(* IEC 61131-3 sources: osaicnc/, 32 files *)

(* ---- F_BitPosition.st ---- *)
(*[[
    UserText1= "V15.7",
]]*)
FUNCTION F_BitPosition : INT
(*
F ***************************************************************************************
F * File name    : F_BitPosition.st                                                     *
F * Description  : Calculate the position of a single bit into the input variable, from *
F *                1 to 15, the function give zero if more then one bit is true, if the *
F *                most significative bit is true, if all the bits are false.           *
F *                Especially thinked to convert the SW31 S_1PROMOD variable in the     *
F *                SetProcessMode function block format.                                *
F ***************************************************************************************
F * Product line : OpenControl                                                          *
F * Enviroment   : PLC Application                                                      *
F * Component    :                                                                      *
F *                                                                                     *
F * ----------------------------------------------------------------------------------- *
F *                                                                                     *
F *   Author        date        comments                                                *
F *                                                                                     *
F *   Mazzocco      19-03-10    Creation F_BitPosition                                  *
F *                                                                                     *
F * ----------------------------------------------------------------------------------- *
F *                                                                                     *
F * Input        :  iiVariable          INT                                             *
F *                     Input variable with only one bit true, except the most          *
F *                     significative bit                                               *
F *                                                                                     *
F * Return       :  INT                                                                 *
F *                     Position of a single bit into the input variable, from 1 to 15, *
F *                     the function give zero if more then one bit or the most         *
F *                     significative bit is true                                       *
F *                                                                                     *
F * Global used  :      Not used                                                        *
F *                                                                                     *
F ***************************************************************************************

	Example for program use

\* F_BitPosition function calculate the position of a single bit into the input variable, from
	1 to 15, the function give zero if more then one bit is true, if the most significative bit
	is true, if all the bits are false */
liNewValue	:= F_BitPosition(iiVariable);
*)

VAR_INPUT
	iiVariable	: int;	(* Input variable with only one bit true, except the most significative bit *)
END_VAR

case iiVariable of
	1:		F_BitPosition	:= 1;
	2:		F_BitPosition	:= 2;
	4:		F_BitPosition	:= 3;
	8:		F_BitPosition	:= 4;
	16:		F_BitPosition	:= 5;
	32:		F_BitPosition	:= 6;
	64:		F_BitPosition	:= 7;
	128:	F_BitPosition	:= 8;
	256:	F_BitPosition	:= 9;
	512:	F_BitPosition	:= 10;
	1024:	F_BitPosition	:= 11;
	2048:	F_BitPosition	:= 12;
	4096:	F_BitPosition	:= 13;
	8192:	F_BitPosition	:= 14;
	16384:	F_BitPosition	:= 15;
	-32768:	F_BitPosition	:= 16;
else
    F_BitPosition	:= 0;
end_case;

END_FUNCTION

(* ---- F_CompareArray.st ---- *)
(*[[
    UserText1= "V15.7",
]]*)
FUNCTION F_CompareArray : BOOL
(*
F ***************************************************************************************
F * File name    : F_CompareArray.st                                                    *
F * Description  : Compare two array with NUM_OF_AX fields, to check if they countain   *
F *                the same value, in the same or in different order.                   *
F ***************************************************************************************
F * Product line : OpenControl                                                          *
F * Enviroment   : PLC Application                                                      *
F * Component    :                                                                      *
F *                                                                                     *
F * ----------------------------------------------------------------------------------- *
F *                                                                                     *
F *   Author        date        comments                                                *
F *                                                                                     *
F *   Mazzocco      18-05-10    Function creation                                       *
F *                                                                                     *
F * ----------------------------------------------------------------------------------- *
F *                                                                                     *
F * Input        :  iiArray1            Array [0..NUM_OF_AX-1] of INT                   *
F *                     First array                                                     *
F *                                                                                     *
F *                 iiArray2            Array [0..NUM_OF_AX-1] of INT                   *
F *                     Second array                                                    *
F *                                                                                     *
F * Return       :  BOOL                                                                *
F *                     True value if both arrays countain the same value in any order  *
F *                                                                                     *
F * Global used  :      Not used                                                        *
F *                                                                                     *
F ***************************************************************************************

	Example for program use

\* Compare two array with NUM_OF_AX fields, to check if they countain the same value, in the
	same or in different order */
lEqual	:= F_CompareArray(iiArray1, iiArray2);
*)

VAR_INPUT
	iiArray1	:Array [0..NUM_OF_AX-1] of int;	(* First array *)
	iiArray2	:Array [0..NUM_OF_AX-1] of int;	(* Second array *)
END_VAR

VAR
	liInd		: int;	(* Array field scrolling *)
END_VAR

for liInd := 0 to (NUM_OF_AX-1) by 1 do

	(* check if the second array countain all the value of the first array *)
	if iiArray1[liInd]=iiArray2[0] or iiArray1[liInd]=iiArray2[1] or
	iiArray1[liInd]=iiArray2[2] or iiArray1[liInd]=iiArray2[3] or
	iiArray1[liInd]=iiArray2[4] or iiArray1[liInd]=iiArray2[5] or
	iiArray1[liInd]=iiArray2[6] or iiArray1[liInd]=iiArray2[7] or
	iiArray1[liInd]=iiArray2[8] or iiArray1[liInd]=iiArray2[9] or
	iiArray1[liInd]=iiArray2[10] or iiArray1[liInd]=iiArray2[11] then
		F_CompareArray	:= true;
	else
		F_CompareArray	:= false;
		exit;
	end_if;

	(* check if the first array countain all the value of the second array *)
	if iiArray2[liInd]=iiArray1[0] or iiArray2[liInd]=iiArray1[1] or
	iiArray2[liInd]=iiArray1[2] or iiArray2[liInd]=iiArray1[3] or
	iiArray2[liInd]=iiArray1[4] or iiArray2[liInd]=iiArray1[5] or
	iiArray2[liInd]=iiArray1[6] or iiArray2[liInd]=iiArray1[7] or
	iiArray2[liInd]=iiArray1[8] or iiArray2[liInd]=iiArray1[9] or
	iiArray2[liInd]=iiArray1[10] or iiArray2[liInd]=iiArray1[11] then
		F_CompareArray	:= true;
	else
		F_CompareArray	:= false;
		exit;
	end_if;

end_for;

END_FUNCTION

(* ---- F_CycleStart.st ---- *)
(*[[
    UserText1= "V15.7",
]]*)
FUNCTION F_CycleStart : DWORD
(*
F ***************************************************************************************
F * File name    : F_CycleStart.st                                                      *
F * Description  : CycleStart request from PLC, works like the system function block    *
F *                with one more flag to decide if the request is comparable to an      *
F *                operator request (like a console) and can be refused by the filter   *
F *                task.                                                                *
F ***************************************************************************************
F * Product line : OpenControl                                                          *
F * Enviroment   : PLC Application                                                      *
F * Component    :                                                                      *
F *                                                                                     *
F * ----------------------------------------------------------------------------------- *
F *                                                                                     *
F *   Author        date        comments                                                *
F *                                                                                     *
F *   Mazzocco      25-11-13    Function creation                                       *
F *                                                                                     *
F * ----------------------------------------------------------------------------------- *
F *                                                                                     *
F * Input        :  iiExecMode          INT                                             *
F *                     Command execution modality: MODE_NOWAIT, MODE_WAIT              *
F *                                                                                     *
F *                 iiProc              INT                                             *
F *                     Process number 1..24                                            *
F *                                                                                     *
F *                 iOpConsole          BOOL                                            *
F *                     Console flag, the request is comparable to an operator console, *
F *                     can be rfeused by filter task                                   *
F *                                                                                     *
F * Return       :  DWORD                                                               *
F *                     CycleStart function block return code                           *
F *                                                                                     *
F * Global used  :  gPlcConCON        array [0..ciMaxProc] of bool                             *
F *                     Cycle start request from Plc console ambient memory             *
F *                                                                                     *
F ***************************************************************************************

	Example for program use

\* CycleStart request from PLC, works like the system function block with two more possibility:
	the request can be applyed to all processes, have one more flag to decide if the request
	is comparable to an operator request (like a console) and can be refused by the filter task. */

llRetCode	:= F_CycleStart(
	iiExecMode,		\* IN	INT		Command execution modality: MODE_NOWAIT, MODE_WAIT */
	iiProc,			\* IN	INT		Process number 1..24 or -1 (ciProcAll) to request to all processes */
	iOpConsole);	\* IN	BOOL	Console flag, the request is comparable to an operator console, can be rfeused by filter task */

\* Example to apply the request only at the selected process with the filter enabled */
llRetCode	:= F_CycleStart(MODE_NOWAIT, SI_PROCSEL, true \*iOpConsole*/);
*)

	#IMPORT  "GvU_Variable.gvl"
	#IMPORT  "Gv_AllProcess.gvl"

VAR_INPUT
	iiExecMode	: int;	(* Command execution modality: MODE_NOWAIT, MODE_WAIT *)
	iiProc		: int;	(* Process number 1..24 or -1 (ciProcAll) to request to all processes *)
	iOpConsole	: bool;	(* Console flag, the request is comparable to an operator console, can be rfeused by filter task *)
END_VAR

VAR
	llExecStatus	: dword;	(* Function block execution status, not used *)
END_VAR;

(* Request for a single process *)
gPlcConCON[iiProc]	:= iOpConsole;	(* Plc console ambient memory *)
F_CycleStart	:= CycleStart(iiExecMode, llExecStatus, iiProc);
if F_CycleStart<>0 then
	gPlcConCON[iiProc]	:= false;	(* In case of error reset the Plc console ambient memory *)
end_if;

END_FUNCTION

(* ---- F_CycleStop.st ---- *)
(*[[
    UserText1= "V15.7",
]]*)
FUNCTION F_CycleStop : DWORD
(*
F ***************************************************************************************
F * File name    : F_CycleStop.st                                                       *
F * Description  : Cycle stop request from PLC, works like the system function block    *
F *                with two more possibility: the request can be applyed to all         *
F *                processes, have one more flag to decide if the request is comparable *
F *                to an operator request (like a console) and can be refused by the    *
F *                filter task.                                                         *
F ***************************************************************************************
F * Product line : OpenControl                                                          *
F * Enviroment   : PLC Application                                                      *
F * Component    :                                                                      *
F *                                                                                     *
F * ----------------------------------------------------------------------------------- *
F *                                                                                     *
F *   Author        date        comments                                                *
F *                                                                                     *
F *   Mazzocco      25-11-13    Function creation                                       *
F *                                                                                     *
F * ----------------------------------------------------------------------------------- *
F *                                                                                     *
F * Input        :  iiExecMode          INT                                             *
F *                     Command execution modality: MODE_NOWAIT, MODE_WAIT              *
F *                                                                                     *
F *                 iiProc              INT                                             *
F *                     Process number 1..24 or -1 (ciProcAll) to request to all        *
F *                     processes.                                                      *
F *                                                                                     *
F *                 iiLastProc          INT                                             *
F *                     Last process number, used only if the request is for all        *
F *                     processes.                                                      *
F *                                                                                     *
F *                 iiNoProc            INT                                             *
F *                     Process number to skip if the request is for all processes,     *
F *                     0 to apply to every processes.                                  *
F *                                                                                     *
F *                 iOpConsole          BOOL                                            *
F *                     Console flag, the request is comparable to an operator console, *
F *                     can be rfeused by filter task                                   *
F *                                                                                     *
F * Return       :  DWORD                                                               *
F *                     CycleStop function block return code                            *
F *                                                                                     *
F * Global used  :  gPlcConCOF          array [0..ciMaxProc] of bool                    *
F *                     Cycle Stop request from Plc console ambient memory              *
F *                                                                                     *
F ***************************************************************************************

	Example for program use

\* Cycle stop request from PLC, works like the system function block with two more possibility:
	the request can be applyed to all processes, have one more flag to decide if the request
	is comparable to an operator request (like a console) and can be refused by the filter task. */

llRetCode	:= F_CycleStop(
	iiExecMode,		\* IN	INT		Command execution modality: MODE_NOWAIT, MODE_WAIT */
	iiProc,			\* IN	INT		Process number 1..24 or -1 (ciProcAll) to request to all processes */
	iiLastProc,		\* IN	INT		Last process number, used only if the request is for all processes */
	iiNoProc,		\* IN	INT		Process number to skip if the request is for all processes, 0 to apply to every processes */
	iOpConsole);	\* IN	BOOL	Console flag, the request is comparable to an operator console, can be rfeused by filter task */

\* Example to apply the request only at the selected process with the filter enabled, the 3rd and 4th input data are not used */
llRetCode	:= F_CycleStop(MODE_NOWAIT, SI_PROCSEL, MI_LastProc, 0 \*iiNoProc*/, true \*iOpConsole*/);

\* Example to apply the request to every existing process with the filter enabled */
llRetCode	:= F_CycleStop(MODE_NOWAIT, ciProcAll, MI_LastProc, 0 \*iiNoProc*/, true \*iOpConsole*/);

\* Example to apply the request to every existing process, except the process number 1, with the filter enabled */
llRetCode	:= F_CycleStop(MODE_NOWAIT, ciProcAll, MI_LastProc, 1 \*iiNoProc*/, true \*iOpConsole*/);
*)

	#IMPORT  "GvU_Variable.gvl"
	#IMPORT  "Gv_Allprocess.gvl"

VAR_INPUT
	iiExecMode	: int;	(* Command execution modality: MODE_NOWAIT, MODE_WAIT *)
	iiProc		: int;	(* Process number 1..24 or -1 (ciProcAll) to request to all processes *)
	iiLastProc	: int;	(* Last process number, used only if the request is for all processes *)
	iiNoProc	: int;	(* Process number to skip, used only if the request is for all processes, 0 to apply to every processes *)
	iOpConsole	: bool;	(* Console flag, the request is comparable to an operator console, can be rfeused by filter task *)
END_VAR

VAR
	llExecStatus	: dword;	(* Function block execution status, not used *)
	liInd			: int;	(* Array index scroll *)
END_VAR;

if iiProc=-1 then	(* Request for all processes *)
	if iiLastProc<1 then
		F_CycleStop	:= 16#00170005;
	end_if;

	for liInd :=1 to iiLastProc by 1 do
		if liInd<>iiNoProc then
			gPlcConCOF[liInd]	:= iOpConsole;	(* Plc console ambient memory *)
			F_CycleStop	:= CycleStop(iiExecMode, llExecStatus, liInd);
			if F_CycleStop<>0 then
				gPlcConCOF[liInd]	:= false;	(* In case of error reset the Plc console ambient memory *)
				exit;
			end_if;
		end_if;
	end_for;
else				(* Request for a single process *)
	gPlcConCOF[iiProc]	:= iOpConsole;	(* Plc console ambient memory *)
	F_CycleStop	:= CycleStop(iiExecMode, llExecStatus, iiProc);
	if F_CycleStop<>0 then
		gPlcConCOF[iiProc]	:= false;	(* In case of error reset the Plc console ambient memory *)
	end_if;
end_if;

END_FUNCTION

(* ---- F_DWordToHexStr.st ---- *)
(*[[
    UserText1= "V15.7",
]]*)
FUNCTION F_DWordToHexStr : STRING
(*
F ***************************************************************************************
F * File name    : F_DWordToHexStr.st                                                   *
F * Description  : Convert a DWORD value into a hexadecimal string                      *
F *                                                                                     *
F ***************************************************************************************
F * Product line : OpenControl                                                          *
F * Enviroment   : PLC Application                                                      *
F * Component    :                                                                      *
F *                                                                                     *
F * ----------------------------------------------------------------------------------- *
F *                                                                                     *
F *   Author        date        comments                                                *
F *                                                                                     *
F *   T. Hall       23-09-12    Function creation                                       *
F *                                                                                     *
F * ----------------------------------------------------------------------------------- *
F *                                                                                     *
F * Input        :  ilInpVal            DWORD                                           *
F *                     Value to convert                                                *
F *                                                                                     *
F *                 iLdgZero            BOOL                                            *
F *                     FALSE=No leading 0's, TRUE=Include leading 0's                  *
F *                                                                                     *
F * Return       :  STRING                                                              *
F *                 String containing the hexadecimal value of ilInpVal                 *
F *                 Depending on the value of iLdgZero leading 0's may be present       *
F *                                                                                     *
F * Global used  :      Not used                                                        *
F *                                                                                     *
F ***************************************************************************************

   Example for program use

\* Convert dword value into hexadecinal string (without leading 0's)
   E.G. 196616 -> '30008' */
MyStr := F_DWordToHexStr( llMyDWrd, FALSE );
*)

VAR_INPUT
   ilInpVal	: dword;  (* Value to convert *)
   iLdgZero : bool;   (* TRUE=return leading 0's *)
END_VAR

VAR
   lChFnd   : bool;
   liShift  : int;
   liChar   : int;
   lsChar   :STRING;
   lsStr    :STRING;
END_VAR

(* Force non-0 found if leading 0's req'd *)
lChFnd := iLdgZero;

(* Loop for 8 chars *)
FOR liShift := 28 TO 0 BY -4 do
   liChar := DWORD_TO_INT( SHR( ilInpVal, liShift ) and 16#F );

   (* Set non-0 found *)
   if liChar <> 0 or liShift = 0 then
      lChFnd := TRUE;
   end_if;

   CASE liChar OF
      10: lsChar := 'A';
      11: lsChar := 'B';
      12: lsChar := 'C';
      13: lsChar := 'D';
      14: lsChar := 'E';
      15: lsChar := 'F';
   else
      lsChar := INT_TO_STRING( liChar );
   END_CASE;

   (* Append Hex char. *)
   if lChFnd then
      lsStr := CONCAT( lsStr, lsChar );
   end_if;

END_FOR;

(* Return Hex string *)
F_DWordToHexStr := lsStr;

END_FUNCTION

(* ---- F_EncodeDword.st ---- *)
(*[[
    UserText1= "V15.7",
]]*)
FUNCTION F_EncodeDword : int

	#IMPORT  "Gv_AllProcess.gvl"

(*
F ***************************************************************************************
F * File name    : F_EncodeDword.st                                                     *
F * Description  : Calculate the position of a single bit into the input variable, from *
F *                1 to 15, the function give zero if more then one bit is true, if the *
F *                most significative bit is true, if all the bits are false.           *
F *                Especially thinked to convert the SW31 S_1PROMOD variable in the     *
F *                SetProcessMode function block format.                                *
F ***************************************************************************************
F * Product line : OpenControl                                                          *
F * Enviroment   : PLC Application                                                      *
F * Component    :                                                                      *
F *                                                                                     *
F * ----------------------------------------------------------------------------------- *
F *                                                                                     *
F *   Author        date        comments                                                *
F *                                                                                     *
F *   Scapolan      19-04-16    Creation F_BitPosition                                  *
F *                                                                                     *
F * ----------------------------------------------------------------------------------- *
F *                                                                                     *
F * Input        :  iiVariable          INT                                             *
F *                     Input variable with only one bit true, except the most          *
F *                     significative bit                                               *
F *                                                                                     *
F * Return       :  INT                                                                 *
F *                     Position of a single bit into the input variable, from 1 to 15, *
F *                     the function give zero if more then one bit or the most         *
F *                     significative bit is true                                       *
F *                                                                                     *
F * Global used  :      Not used                                                        *
F *                                                                                     *
F ***************************************************************************************

	Example for program use

\* F_BitPosition function calculate the position of a single bit into the input variable, from
	1 to 15, the function give zero if more then one bit is true, if the most significative bit
	is true, if all the bits are false */
liNewValue	:= F_BitPosition(iiVariable);
*)

VAR_INPUT
	il_Variable	: dword;	(* Input variable with only one bit true, except the most significative bit *)
END_VAR

var
	li_Position	: int;
	ll_RetCode	: dword;
end_var

ll_RetCode := SearchData(0, 33, il_Variable, GL_varfound[0], li_Position);
if li_Position = -1 then
	F_EncodeDword := 0;
else
	F_EncodeDword := li_Position;
end_if;

END_FUNCTION

(* ---- F_Gestop_Close.st ---- *)
(*[[
    UserText1= "V15.7",
]]*)
(*
F *******************************************************************************************
F * File name	: F_Gestop_Close.st															*
F * Description	: request the EMERGENCYSTOPCLOSE and set to one the configured fast output	*
F *******************************************************************************************
F * Product line : OpenControl                                                          	*
F * Enviroment   : PLC Application                                                      	*
F * Component    :                                                                      	*
F * ----------------------------------------------------------------------------------------*
F *   Author        date        comments                                                	*
F *   Scapolan      19-05-16    Function creation                                       	*
F * ----------------------------------------------------------------------------------------*
F * Input        :	none																	*
F *******************************************************************************************
*)

FUNCTION F_Gestop_Close

	#IMPORT  "Gv_AllProcess.gvl"
	#IMPORT  "Gv_InputOutput.gvl"

var
	li_FastOutStatus	: word;
	ll_RetCode			: dword;
end_var

(* Close the emergency contact - fast output 1 *)
ll_Retcode := EmergencyStopClose(0);

if (gSt_PlcCfg.Second_Estop_Signal <> 0) then
	if (gSt_PlcCfg.Second_Estop_Signal > 0) and (gSt_PlcCfg.Second_Estop_Signal < 4) then
		li_FastOutStatus := SHL(1, gSt_PlcCfg.Second_Estop_Signal-1);
		ll_RetCode	:= FastOutputWrite(li_FastOutStatus, li_FastOutStatus);
	end_if;
end_if;

O_AuxGestop := 1;
M_SpepnOpen	:= false;

END_FUNCTION

(* ---- F_Gestop_Open.st ---- *)
(*[[
    UserText1= "V15.7",
]]*)
(*
F *******************************************************************************************
F * File name	: F_Gestop_Open.st															*
F * Description	: request the EMERGENCYSTOPOPEN and set to ZERO the configured fast output	*
F *******************************************************************************************
F * Product line : OpenControl                                                          	*
F * Enviroment   : PLC Application                                                      	*
F * Component    :                                                                      	*
F * ----------------------------------------------------------------------------------------*
F *   Author        date        comments                                                	*
F *   Scapolan      19-05-16    Function creation                                       	*
F * ----------------------------------------------------------------------------------------*
F * Input        :	none																	*
F *******************************************************************************************
*)
FUNCTION F_Gestop_Open

	#IMPORT  "Gv_AllProcess.gvl"
	#IMPORT  "Gv_InputOutput.gvl"

var
	li_OutMask			: word;
	ll_RetCode			: dword;
end_var

(* Open the emergency contact - fast output 1 = 0 *)
ll_RetCode := EmergencyStopOpen(0, 0);

if (gSt_PlcCfg.Second_Estop_Signal <> 0) then
	if (gSt_PlcCfg.Second_Estop_Signal > 0) and (gSt_PlcCfg.Second_Estop_Signal < 4) then
		li_OutMask := SHL(1, gSt_PlcCfg.Second_Estop_Signal-1);
		ll_RetCode	:= FastOutputWrite(0, li_OutMask);
	end_if;
end_if;

O_AuxGestop := 0;
M_SpepnOpen	:= true;
I_AuxOn := false;

END_FUNCTION

(* ---- F_Get_Sys_Type.st ---- *)
(*[[
    UserText1= "V15.7",
]]*)
FUNCTION F_Get_Sys_Type
	#IMPORT  "Gv_AllProcess.gvl"

var
	ll_RetCode			: dword;
	lb_Board_type		: byte;						(* Board type code *)
end_var

	(* Get current board of system, the system can use max 2 board 0 and 1 *)
	(* Board 0 *)
	ll_RetCode := GetBoardInfo(0, gSt_BoardInfo_0);
	lb_Board_type := Dword_to_byte(SHR(gSt_BoardInfo_0.BusDescr1, 8));
	if    (lb_Board_type = DGT_BUS_SERCOS) 			then gBoard_0_DGT_BUS_SERCOS 		:= true;
	elsif (lb_Board_type = DGT_BUS_MECHATROLINK)	then gBoard_0_DGT_BUS_MECHATROLINK	:= true;
	elsif (lb_Board_type = DGT_BUS_OSWIRE)			then gBoard_0_DGT_BUS_OSWIRE		:= true;
	elsif (lb_Board_type = DGT_BUS_CANOPEN)			then gBoard_0_DGT_BUS_CANOPEN		:= true;
	elsif (lb_Board_type = DGT_BUS_PROFIBUS)		then gBoard_0_DGT_BUS_PROFIBUS		:= true;
	elsif (lb_Board_type = DGT_BUS_ETN)				then gBoard_0_DGT_BUS_ETN			:= true;
	elsif (lb_Board_type = DGT_BUS_ETHERCAT)		then gBoard_0_DGT_BUS_ETHERCAT		:= true;
	end_if;

	lb_Board_type := Dword_to_byte(SHR(gSt_BoardInfo_0.BusDescr2, 8));
	if    (lb_Board_type = DGT_BUS_SERCOS) 			then gBoard_0_DGT_BUS_SERCOS 		:= true;
	elsif (lb_Board_type = DGT_BUS_MECHATROLINK)	then gBoard_0_DGT_BUS_MECHATROLINK	:= true;
	elsif (lb_Board_type = DGT_BUS_OSWIRE)			then gBoard_0_DGT_BUS_OSWIRE		:= true;
	elsif (lb_Board_type = DGT_BUS_CANOPEN)			then gBoard_0_DGT_BUS_CANOPEN		:= true;
	elsif (lb_Board_type = DGT_BUS_PROFIBUS)		then gBoard_0_DGT_BUS_PROFIBUS		:= true;
	elsif (lb_Board_type = DGT_BUS_ETN)				then gBoard_0_DGT_BUS_ETN			:= true;
	elsif (lb_Board_type = DGT_BUS_ETHERCAT)		then gBoard_0_DGT_BUS_ETHERCAT		:= true;
	end_if;

	lb_Board_type := Dword_to_byte(SHR(gSt_BoardInfo_0.BusDescr3, 8));
	if    (lb_Board_type = DGT_BUS_SERCOS) 			then gBoard_0_DGT_BUS_SERCOS 		:= true;
	elsif (lb_Board_type = DGT_BUS_MECHATROLINK)	then gBoard_0_DGT_BUS_MECHATROLINK	:= true;
	elsif (lb_Board_type = DGT_BUS_OSWIRE)			then gBoard_0_DGT_BUS_OSWIRE		:= true;
	elsif (lb_Board_type = DGT_BUS_CANOPEN)			then gBoard_0_DGT_BUS_CANOPEN		:= true;
	elsif (lb_Board_type = DGT_BUS_PROFIBUS)		then gBoard_0_DGT_BUS_PROFIBUS		:= true;
	elsif (lb_Board_type = DGT_BUS_ETN)				then gBoard_0_DGT_BUS_ETN			:= true;
	elsif (lb_Board_type = DGT_BUS_ETHERCAT)		then gBoard_0_DGT_BUS_ETHERCAT		:= true;
	end_if;

	lb_Board_type := Dword_to_byte(SHR(gSt_BoardInfo_0.BusDescr4, 8));
	if    (lb_Board_type = DGT_BUS_SERCOS) 			then gBoard_0_DGT_BUS_SERCOS 		:= true;
	elsif (lb_Board_type = DGT_BUS_MECHATROLINK)	then gBoard_0_DGT_BUS_MECHATROLINK	:= true;
	elsif (lb_Board_type = DGT_BUS_OSWIRE)			then gBoard_0_DGT_BUS_OSWIRE		:= true;
	elsif (lb_Board_type = DGT_BUS_CANOPEN)			then gBoard_0_DGT_BUS_CANOPEN		:= true;
	elsif (lb_Board_type = DGT_BUS_PROFIBUS)		then gBoard_0_DGT_BUS_PROFIBUS		:= true;
	elsif (lb_Board_type = DGT_BUS_ETN)				then gBoard_0_DGT_BUS_ETN			:= true;
	elsif (lb_Board_type = DGT_BUS_ETHERCAT)		then gBoard_0_DGT_BUS_ETHERCAT		:= true;
	end_if;

	(* Board 1 *)
	ll_RetCode := GetBoardInfo(1, gSt_BoardInfo_1);
	lb_Board_type := Dword_to_byte(SHR(gSt_BoardInfo_1.BusDescr1, 8));
	if    (lb_Board_type = DGT_BUS_SERCOS) 			then gBoard_1_DGT_BUS_SERCOS 		:= true;
	elsif (lb_Board_type = DGT_BUS_MECHATROLINK)	then gBoard_1_DGT_BUS_MECHATROLINK	:= true;
	elsif (lb_Board_type = DGT_BUS_OSWIRE)			then gBoard_1_DGT_BUS_OSWIRE		:= true;
	elsif (lb_Board_type = DGT_BUS_CANOPEN)			then gBoard_1_DGT_BUS_CANOPEN		:= true;
	elsif (lb_Board_type = DGT_BUS_PROFIBUS)		then gBoard_1_DGT_BUS_PROFIBUS		:= true;
	elsif (lb_Board_type = DGT_BUS_ETN)				then gBoard_1_DGT_BUS_ETN			:= true;
	elsif (lb_Board_type = DGT_BUS_ETHERCAT)		then gBoard_1_DGT_BUS_ETHERCAT		:= true;
	end_if;

	lb_Board_type := Dword_to_byte(SHR(gSt_BoardInfo_1.BusDescr2, 8));
	if    (lb_Board_type = DGT_BUS_SERCOS) 			then gBoard_1_DGT_BUS_SERCOS 		:= true;
	elsif (lb_Board_type = DGT_BUS_MECHATROLINK)	then gBoard_1_DGT_BUS_MECHATROLINK	:= true;
	elsif (lb_Board_type = DGT_BUS_OSWIRE)			then gBoard_1_DGT_BUS_OSWIRE		:= true;
	elsif (lb_Board_type = DGT_BUS_CANOPEN)			then gBoard_1_DGT_BUS_CANOPEN		:= true;
	elsif (lb_Board_type = DGT_BUS_PROFIBUS)		then gBoard_1_DGT_BUS_PROFIBUS		:= true;
	elsif (lb_Board_type = DGT_BUS_ETN)				then gBoard_1_DGT_BUS_ETN			:= true;
	elsif (lb_Board_type = DGT_BUS_ETHERCAT)		then gBoard_1_DGT_BUS_ETHERCAT		:= true;
	end_if;

	lb_Board_type := Dword_to_byte(SHR(gSt_BoardInfo_1.BusDescr3, 8));
	if    (lb_Board_type = DGT_BUS_SERCOS) 			then gBoard_1_DGT_BUS_SERCOS 		:= true;
	elsif (lb_Board_type = DGT_BUS_MECHATROLINK)	then gBoard_1_DGT_BUS_MECHATROLINK	:= true;
	elsif (lb_Board_type = DGT_BUS_OSWIRE)			then gBoard_1_DGT_BUS_OSWIRE		:= true;
	elsif (lb_Board_type = DGT_BUS_CANOPEN)			then gBoard_1_DGT_BUS_CANOPEN		:= true;
	elsif (lb_Board_type = DGT_BUS_PROFIBUS)		then gBoard_1_DGT_BUS_PROFIBUS		:= true;
	elsif (lb_Board_type = DGT_BUS_ETN)				then gBoard_1_DGT_BUS_ETN			:= true;
	elsif (lb_Board_type = DGT_BUS_ETHERCAT)		then gBoard_1_DGT_BUS_ETHERCAT		:= true;
	end_if;

	lb_Board_type := Dword_to_byte(SHR(gSt_BoardInfo_1.BusDescr4, 8));
	if    (lb_Board_type = DGT_BUS_SERCOS) 			then gBoard_1_DGT_BUS_SERCOS 		:= true;
	elsif (lb_Board_type = DGT_BUS_MECHATROLINK)	then gBoard_1_DGT_BUS_MECHATROLINK	:= true;
	elsif (lb_Board_type = DGT_BUS_OSWIRE)			then gBoard_1_DGT_BUS_OSWIRE		:= true;
	elsif (lb_Board_type = DGT_BUS_CANOPEN)			then gBoard_1_DGT_BUS_CANOPEN		:= true;
	elsif (lb_Board_type = DGT_BUS_PROFIBUS)		then gBoard_1_DGT_BUS_PROFIBUS		:= true;
	elsif (lb_Board_type = DGT_BUS_ETN)				then gBoard_1_DGT_BUS_ETN			:= true;
	elsif (lb_Board_type = DGT_BUS_ETHERCAT)		then gBoard_1_DGT_BUS_ETHERCAT		:= true;
	end_if;

END_FUNCTION

(* ---- F_HoldOFF.st ---- *)
(*[[
    UserText1= "V15.7",
]]*)
FUNCTION F_HoldOFF : DWORD
(*
F ***************************************************************************************
F * File name    : F_HoldOFF.st                                                         *
F * Description  : Hold OFF request from PLC, works like the system function block with *
F *                two more possibility: the request can be applyed to all processes,   *
F *                have one more flag to decide if the request is comparable to an      *
F *                operator request (like a console) and can be refused by the filter   *
F *                task.                                                                *
F ***************************************************************************************
F * Product line : OpenControl                                                          *
F * Enviroment   : PLC Application                                                      *
F * Component    :                                                                      *
F *                                                                                     *
F * ----------------------------------------------------------------------------------- *
F *                                                                                     *
F *   Author        date        comments                                                *
F *                                                                                     *
F *   Scapolan      06-07-16    Function creation                                       *
F *                                                                                     *
F * ----------------------------------------------------------------------------------- *
F *                                                                                     *
F * Input        :  iiProc              INT                                             *
F *                     Process number 1..24 or -1 (ciProcAll) to request to all        *
F *                     processes.                                                      *
F *                                                                                     *
F *                 iOpConsole          BOOL                                            *
F *                     Console flag, the request is comparable to an operator console, *
F *                     can be rfeused by filter task                                   *
F *                                                                                     *
F * Return       :  DWORD                                                               *
F *                     HoldOFF function block return code                              *
F *                                                                                     *
F * Global used  :  gPlcConHOF          array [0..ciMaxProc] of bool                    *
F *                     HoldOFF request from Plc console ambient memory                 *
F *                                                                                     *
F ***************************************************************************************

	Example for program use

\* Hold OFF request from PLC, works like the system function block with two more possibility:
	the request can be applyed to all processes, have one more flag to decide if the request
	is comparable to an operator request (like a console) and can be refused by the filter task. */

llRetCode	:= F_HoldOFF(
	iiProc,			\* IN	INT		Process number 1..24 or -1 (ciProcAll) to request to all processes */
	iOpConsole);	\* IN	BOOL	Console flag, the request is comparable to an operator console, can be rfeused by filter task */

\* Example to apply the request to every existing process, with the filter enabled */
llRetCode	:= F_HoldOFF(ciProc, true \*iOpConsole*/);
*)

	#IMPORT  "GvU_Variable.gvl"
	#IMPORT  "Gv_Allprocess.gvl"

VAR_INPUT
	iiProc		: int;	(* Process number 1..24 or -1 (ciProcAll) to request to all processes *)
	iOpConsole	: bool;	(* Console flag, the request is comparable to an operator console, can be rfeused by filter task *)
END_VAR

VAR
	llExecStatus	: dword;	(* Function block execution status, not used *)
END_VAR;

gPlcConHOF[iiProc]	:= iOpConsole;	(* Plc console ambient memory *)
F_HoldOFF	:= HoldOFF(MODE_NOWAIT, llExecStatus, iiProc);

END_FUNCTION

(* ---- F_HoldON.st ---- *)
(*[[
    UserText1= "V15.7",
]]*)
FUNCTION F_HoldON : DWORD
(*
F ***************************************************************************************
F * File name    : F_HoldON.st                                                          *
F * Description  : Hold ON request from PLC, works like the system function block with  *
F *                two more possibility: the request can be applyed to all processes,   *
F *                have one more flag to decide if the request is comparable to an      *
F *                operator request (like a console) and can be refused by the filter   *
F *                task.                                                                *
F ***************************************************************************************
F * Product line : OpenControl                                                          *
F * Enviroment   : PLC Application                                                      *
F * Component    :                                                                      *
F *                                                                                     *
F * ----------------------------------------------------------------------------------- *
F *                                                                                     *
F *   Author        date        comments                                                *
F *                                                                                     *
F *   Scapolan		06-07-16    Function creation                                       *
F *                                                                                     *
F * ----------------------------------------------------------------------------------- *
F *                                                                                     *
F * Input        :  iiExecMode          INT                                             *
F *                     Command execution modality: MODE_NOWAIT, MODE_WAIT              *
F *                                                                                     *
F *                 iiProc              INT                                             *
F *                     Process number 1..24 or -1 (ciProcAll) to request to all        *
F *                     processes.                                                      *
F *                                                                                     *
F *                 iiLastProc          INT                                             *
F *                     Last process number, used only if the request is for all        *
F *                     processes.                                                      *
F *                                                                                     *
F *                 iiNoProc            INT                                             *
F *                     Process number to skip if the request is for all processes,     *
F *                     0 to apply to every processes.                                  *
F *                                                                                     *
F *                 iOpConsole          BOOL                                            *
F *                     Console flag, the request is comparable to an operator console, *
F *                     can be rfeused by filter task                                   *
F *                                                                                     *
F * Return       :  DWORD                                                               *
F *                     HoldON function block return code                               *
F *                                                                                     *
F * Global used  :  gPlcConHON          array [0..ciMaxProc] of bool                    *
F *                     HoldON request from Plc console ambient memory                  *
F *                                                                                     *
F ***************************************************************************************

	Example for program use

\* Hold ON request from PLC, works like the system function block with two more possibility:
	the request can be applyed to all processes, have one more flag to decide if the request
	is comparable to an operator request (like a console) and can be refused by the filter task. */

llRetCode	:= F_HoldON(
	iiExecMode,		\* IN	INT		Command execution modality: MODE_NOWAIT, MODE_WAIT */
	iiProc,			\* IN	INT		Process number 1..24 or -1 (ciProcAll) to request to all processes */
	iiLastProc,		\* IN	INT		Last process number, used only if the request is for all processes */
	iiNoProc,		\* IN	INT		Process number to skip if the request is for all processes, 0 to apply to every processes */
	iOpConsole);	\* IN	BOOL	Console flag, the request is comparable to an operator console, can be rfeused by filter task */

\* Example to apply the request only at the selected process with the filter enabled, the 3rd and 4th input data are not used */
llRetCode	:= F_HoldON(MODE_NOWAIT, SI_PROCSEL, MI_LastProc, 0 \*iiNoProc*/, true \*iOpConsole*/);

\* Example to apply the request to every existing process with the filter enabled */
llRetCode	:= F_HoldON(MODE_NOWAIT, ciProcAll, MI_LastProc, 0 \*iiNoProc*/, true \*iOpConsole*/);

\* Example to apply the request to every existing process, except the process number 1, with the filter enabled */
llRetCode	:= F_HoldON(MODE_NOWAIT, ciProcAll, MI_LastProc, 1 \*iiNoProc*/, true \*iOpConsole*/);
*)

	#IMPORT  "GvU_Variable.gvl"
	#IMPORT  "Gv_Allprocess.gvl"

VAR_INPUT
	iiProc		: int;	(* Process number 1..24 or -1 (ciProcAll) to request to all processes *)
	iOpConsole	: bool;	(* Console flag, the request is comparable to an operator console, can be rfeused by filter task *)
END_VAR

VAR
	llExecStatus	: dword;	(* Function block execution status, not used *)
END_VAR;

gPlcConHON[iiProc]	:= iOpConsole;	(* Plc console ambient memory *)
F_HoldON	:= HoldON(MODE_NOWAIT, llExecStatus, iiProc);

END_FUNCTION

(* ---- F_Override.st ---- *)
(*[[
    UserText1= "V15.7",
]]*)
FUNCTION F_Override : INT
(*
F ***************************************************************************************
F * File name    : F_Override.st                                                        *
F * Description  : Calculate the new override, compare the requested value with the     *
F *                default array, and find the nearest value                            *
F ***************************************************************************************
F * Product line : OpenControl                                                          *
F * Enviroment   : PLC Application                                                      *
F * Component    :                                                                      *
F *                                                                                     *
F * ----------------------------------------------------------------------------------- *
F *                                                                                     *
F *   Author        date        comments                                                *
F *                                                                                     *
F *   Mazzocco      18-03-10    Creation F_Override                                     *
F *                                                                                     *
F * ----------------------------------------------------------------------------------- *
F *                                                                                     *
F * Input        :  iiValue             array [0..100] of INT                           *
F *                     Default override value array                                    *
F *                                                                                     *
F *                 iiIndMax            INT                                             *
F *                     Maximum array index (min 1, max "ciMaxOvr" constant), is the    *
F *                     number of desired override value                                *
F *                                                                                     *
F *                 iiActValue          INT                                             *
F *                     Actual override value                                           *
F *                                                                                     *
F *                 iiNewValue          INT                                             *
F *                     New override value requested                                    *
F *                                                                                     *
F * Return       :  INT                                                                 *
F *                     New override value, the nearest value at the request searching  *
F *                     into the default array                                          *
F *                                                                                     *
F * Global used  :      Not used                                                        *
F *                                                                                     *
F * Constant used:  ciMaxOvr            INT                                             *
F *                     To knows the dimension of output array used field               *
F *                                                                                     *
F ***************************************************************************************

	Example for program use

\* Calculate the new override, compare the requested value with the default array, and find the
	nearest value */
liNewValue	:= F_Override(
	iiValue,		\* IN	array INT	Default override value array */
	iiIndMax,		\* IN	INT			Maximum array index (min 1, max "ciMaxOvr" constant), is the number of desired override value */
	iiActValue,		\* IN	INT			Actual override value */
	iiNewValue);	\* IN	INT			New override value requested *)

VAR_INPUT
	iiValue		: array [0..ciMaxOvr] of int;	(* Default override value array *)
	iiIndMax	: int;	(* Maximum array index (min 1, max "ciMaxOvr" constant), is the number of desired override value *)
	iiActValue	: int;	(* Actual override value *)
	iiNewValue	: int;	(* New override value requested *)
END_VAR

VAR
	liIndMax	: int;	(* Maximum array index copy *)
	liInd		: int;	(* Index to scroll the array *)
	liActInd	: int;	(* Actual override value index *)
	liPreInd	: int;	(* New override value index precalculated *)
	liNewInd	: int;	(* New override value index *)
END_VAR

(* Check the maximum array index value *)
liIndMax	:= LIMIT(0, iiIndMax, ciMaxOvr);

(* Search into array the nearest value at the actual value to refresh actual index, is
	necessary if the override can be changed from different ambient *)
for liInd := 0 to liIndMax by 1 do
	if iiValue[liInd] <= iiActValue then
		liActInd	:= liInd;
	else
		(* When the next index override value become bigger of the actual value, exit from the
			for cycle, in this way the override index stored is equal or a little bit lowest of
			the actual override value *)
		exit;
	end_if;
end_for;

(* Calculate the new array index *)
if iiNewValue > iiActValue then
	liPreInd	:= liActInd + 1;
elsif iiNewValue < iiActValue then
	liPreInd	:= liActInd - 1;
else
	liPreInd	:= liActInd;
end_if;

(* Check the new index value *)
liNewInd	:= LIMIT(0, liPreInd, liIndMax);

(* Calculate the new override value *)
F_Override	:= iiValue[liNewInd];

END_FUNCTION

(* ---- F_R_TRIG.st ---- *)
(*[[
    UserText1= "V15.7",
]]*)
FUNCTION F_R_TRIG	: bool

VAR_INPUT
	ii_Input	: bool;
END_VAR

VAR_IN_OUT
	ii_Memory	: bool;
END_VAR

if ii_Input and not ii_Memory then
	F_R_TRIG	:= true;
else
	F_R_TRIG	:= false;
end_if;

ii_Memory := ii_Input;

END_FUNCTION

(* ---- F_Reset.st ---- *)
(*[[
    UserText1= "V15.7",
]]*)
FUNCTION F_Reset : DWORD
(*
F ***************************************************************************************
F * File name    : F_Reset.st                                                           *
F * Description  : Reset request from PLC, works like the system function block with    *
F *                two more possibility: the request can be applyed to all processes,   *
F *                have one more flag to decide if the request is comparable to an      *
F *                operator request (like a console) and can be refused by the filter   *
F *                task.                                                                *
F ***************************************************************************************
F * Product line : OpenControl                                                          *
F * Enviroment   : PLC Application                                                      *
F * Component    :                                                                      *
F *                                                                                     *
F * ----------------------------------------------------------------------------------- *
F *                                                                                     *
F *   Author        date        comments                                                *
F *                                                                                     *
F *   Scapolan      06-07-16    Function creation                                       *
F *                                                                                     *
F * ----------------------------------------------------------------------------------- *
F *                                                                                     *
F * Input        :  iiExecMode          INT                                             *
F *                     Command execution modality: MODE_NOWAIT, MODE_WAIT              *
F *                                                                                     *
F *                 iiProc              INT                                             *
F *                     Process number 1..24 or -1 (ciProcAll) to request to all        *
F *                     processes.                                                      *
F *                                                                                     *
F *                 iiLastProc          INT                                             *
F *                     Last process number, used only if the request is for all        *
F *                     processes.                                                      *
F *                                                                                     *
F *                 iiNoProc            INT                                             *
F *                     Process number to skip if the request is for all processes,     *
F *                     0 to apply to every processes.                                  *
F *                                                                                     *
F *                 iOpConsole          BOOL                                            *
F *                     Console flag, the request is comparable to an operator console, *
F *                     can be rfeused by filter task                                   *
F *                                                                                     *
F * Return       :  DWORD                                                               *
F *                     Reset function block return code                                *
F *                                                                                     *
F * Global used  :  gPlcConReset        array [0..ciMaxProc] of bool                    *
F *                     Reset request from Plc console ambient memory                   *
F *                                                                                     *
F ***************************************************************************************

	Example for program use

\* Reset request from PLC, works like the system function block with two more possibility:
	the request can be applyed to all processes, have one more flag to decide if the request
	is comparable to an operator request (like a console) and can be refused by the filter task. */

llRetCode	:= F_Reset(
	iiExecMode,		\* IN	INT		Command execution modality: MODE_NOWAIT, MODE_WAIT */
	iiProc,			\* IN	INT		Process number 1..24 or -1 (ciProcAll) to request to all processes */
	iiLastProc,		\* IN	INT		Last process number, used only if the request is for all processes */
	iiNoProc,		\* IN	INT		Process number to skip if the request is for all processes, 0 to apply to every processes */
	iOpConsole);	\* IN	BOOL	Console flag, the request is comparable to an operator console, can be rfeused by filter task */

\* Example to apply the request only at the selected process with the filter enabled, the 3rd and 4th input data are not used */
llRetCode	:= F_Reset(MODE_NOWAIT, SI_PROCSEL, MI_LastProc, 0 \*iiNoProc*/, true \*iOpConsole*/);

\* Example to apply the request to every existing process with the filter enabled */
llRetCode	:= F_Reset(MODE_NOWAIT, ciProcAll, MI_LastProc, 0 \*iiNoProc*/, true \*iOpConsole*/);

\* Example to apply the request to every existing process, except the process number 1, with the filter enabled */
llRetCode	:= F_Reset(MODE_NOWAIT, ciProcAll, MI_LastProc, 1 \*iiNoProc*/, true \*iOpConsole*/);
*)

	#IMPORT  "GvU_Variable.gvl"
	#IMPORT  "Gv_AllProcess.gvl"

VAR_INPUT
	iiProc		: int;	(* Process number 1..24 or -1 (ciProcAll) to request to all processes *)
	iOpConsole	: bool;	(* Console flag, the request is comparable to an operator console, can be rfeused by filter task *)
END_VAR

VAR
	llExecStatus	: dword;	(* Function block execution status, not used *)
END_VAR;

gPlcConReset[iiProc]	:= iOpConsole;	(* Plc console ambient memory *)
F_Reset	:= Reset(MODE_NOWAIT, llExecStatus, iiProc);

END_FUNCTION

(* ---- F_ReturnCode.st ---- *)
(*[[
    UserText1= "V15.7",
]]*)
FUNCTION F_ReturnCode : DWORD
(*
F ***************************************************************************************
F * File name    : F_ReturnCode.st                                                      *
F * Description  : Function block return code management, save into the system history  *
F *                the return code value, the function block and the program name.      *
F *                Return in output the last saved code, to don't save another time the *
F *                same error.                                                          *
F ***************************************************************************************
F * Product line : OpenControl                                                          *
F * Enviroment   : PLC Application                                                      *
F * Component    :                                                                      *
F *                                                                                     *
F * ----------------------------------------------------------------------------------- *
F *                                                                                     *
F *   Author        date        comments                                                *
F *                                                                                     *
F *   Mazzocco      27-03-14    Function creation                                       *
F *   Scapolan      16-06-16    Optimization                                            *
F *                                                                                     *
F * ----------------------------------------------------------------------------------- *
F *                                                                                     *
F * Input        :  illRetCode          DWORD                                           *
F *                     Function block return code                                      *
F *                                                                                     *
F *                 iaaFBName           STRING                                          *
F *                     Function block name                                             *
F *                                                                                     *
F *                 iaaProgName         STRING                                          *
F *                     Program name                                                    *
F *                                                                                     *
F * Input/Output :  ioMsg               BOOL                                            *
F *                     Generic function block anomaly message                          *
F *                                                                                     *
F * Return       :  DWORD                                                               *
F *                     Last saved code, to don't save another time the same error      *
F *                                                                                     *
F * Global used  :  not used                                                            *
F *                                                                                     *
F ***************************************************************************************

	Example for program use

\* Function block return code management, save into the system history the return code value,
	the function block and the program name. Return in output the last saved code, to don't
	save another time the same error. */

if llRetCode01<>illRetCode then
	llRetCode01	:= F_ReturnCode(
		illRetCode,		\* IN	DWORD	Function block return code */
		iaaFBName,		\* IN	STRING	Function block name */
		iaaProgName,	\* IN	STRING	Program name */
		ioMsg);			\* I/O	BOOL	Generic function block anomaly message */
end_if;

VAR
	laaProgName	:STRING	:= '';	\* Program name */
	llRetCode01	: dword;	\* Return code management */
END_VAR

if llRetCode01<>llRetCode then
	llRetCode01	:= F_ReturnCode(llRetCode, 'iaaFBName', laaProgName, M_Msg);
end_if;
*)

VAR_INPUT
	illRetCode	: dword;		(* Function block return code *)
	iaaFBName	:STRING;	(* Function block name *)
	iaaProgName	:STRING;	(* Program name *)
END_VAR

VAR_IN_OUT
	ioMsg	: bool;	(* Generic function block anomaly message *)
END_VAR

VAR
	laaMessage		:STRING;	(* MEssage saved in system history *)
	llRetCode		: dword;		(* Warning message function block return code *)
END_VAR

if illRetCode<>0 then
	(* Build the message *)
	laaMessage	:= CONCAT(
							'99-Generic FB anomaly, Code: ',
					    	DWORD_TO_STRING(illRetCode),
					    	', Function: ',
					    	iaaFBName,
					   		', Program: ',
							iaaProgName
						 );

	(* Write message into the system history *)
	llRetCode	:= WarningMessage(laaMessage, 1 (*OnHistory*));

	(* Visualize the standard message *)
	ioMsg	:= true;
end_if;

F_ReturnCode	:= illRetCode;

END_FUNCTION

(* ---- F_SetFeedOverride.st ---- *)
(*[[
    UserText1= "V15.7",
]]*)
FUNCTION F_SetFeedOverride : DWORD
(*
F ***************************************************************************************
F * File name    : F_SetFeedOverride.st                                                 *
F * Description  : Set Feed override request from PLC, works like the system function   *
F *                block with three more possibility: the request can be applyed to all *
F *                processes, one flag permit to decide if the request is comparable    *
F *                to an operator request (like a console) and can be refused by the    *
F *                filter task, another flag enable the modification of the override    *
F *                value in the filter task (for example to align at the predefined     *
F *                steps).                                                              *
F ***************************************************************************************
F * Product line : OpenControl                                                          *
F * Enviroment   : PLC Application                                                      *
F * Component    :                                                                      *
F *                                                                                     *
F * ----------------------------------------------------------------------------------- *
F *                                                                                     *
F *   Author        date        comments                                                *
F *                                                                                     *
F *   Scapolan      19-05-16    Function creation                                       *
F *                                                                                     *
F * ----------------------------------------------------------------------------------- *
F *                                                                                     *
F * Input        :  iiExecMode          INT                                             *
F *                     Command execution modality: MODE_NOWAIT, MODE_WAIT              *
F *                                                                                     *
F *                 iiProc              INT                                             *
F *                     Process number 1..24 or -1 (ciProcAll) to request to all        *
F *                     processes.                                                      *
F *                                                                                     *
F *                 iiLastProc          INT                                             *
F *                     Last process number, used only if the request is for all        *
F *                     processes.                                                      *
F *                                                                                     *
F *                 iiNoProc            INT                                             *
F *                     Process number to skip if the request is for all processes,     *
F *                     0 to apply to every processes.                                  *
F *                                                                                     *
F *                 iiPercent           INT                                             *
F *                     New override value 10000=100%                                   *
F *                                                                                     *
F *                 iOpConsole          BOOL                                            *
F *                     Console flag, the request is comparable to an operator console, *
F *                     can be rfeused by filter task                                   *
F *                                                                                     *
F *                 iOpAdjust           BOOL                                            *
F *                     Enable modification (Adjust) of override value from PLC request *
F *                                                                                     *
F * Return       :  DWORD                                                               *
F *                     SetFeedOverride function block return code                      *
F *                                                                                     *
F * Global used  :  gPlcConOvrF          array [0..ciMaxProc] of bool                   *
F *                     Set Feed override request from Plc console ambient memory       *
F *                                                                                     *
F *                 gPlcConAdjF          array [0..ciMaxProc] of BOOL                   *
F *                     Enable the modification of the override value in the filter     *
F *                     task (for example to align at the predefined steps)             *
F *                                                                                     *
F ***************************************************************************************

	Example for program use

\* Set Feed override request from PLC, works like the system function block with two more possibility:
	the request can be applyed to all processes, one flag permit to decide if the request is comparable
	to an operator request (like a console) and can be refused by the filter task, another flag enable the
	modification of the override value in the filter task (for example to align at the predefined steps). */

llRetCode	:= F_SetFeedOverride(
	iiExecMode,		\* IN	INT		Command execution modality: MODE_NOWAIT, MODE_WAIT */
	iiProc,			\* IN	INT		Process number 1..24 or -1 (ciProcAll) to request to all processes */
	iiLastProc,		\* IN	INT		Last process number, used only if the request is for all processes */
	iiNoProc,		\* IN	INT		Process number to skip if the request is for all processes, 0 to apply to every processes */
	iiPercent,		\* IN	INT		New override value 10000=100% */
	iOpConsole,		\* IN	BOOL	Console flag, the request is comparable to an operator console, can be rfeused by filter task */
	iOpAdjust);		\* IN	BOOL	Enable modification (Adjust) of override value from this PLC request */

\* Example to apply the request only at the selected process with the filter enabled, the 3rd and 4th input data are not used,
	the override value are not modified in the filter task */
llRetCode	:= F_SetFeedOverride(MODE_NOWAIT, SI_PROCSEL, MI_LastProc, 0 \*iiNoProc*/, liOverride, true \*iOpConsole*/, false \*iOpAdjust*/);

\* Example to apply the request to every existing process with the filter enabled,
	but the override value are not modified in the filter task */
llRetCode	:= F_SetFeedOverride(MODE_NOWAIT, ciProcAll, MI_LastProc, 0 \*iiNoProc*/, liOverride, true \*iOpConsole*/, false \*iOpAdjust*/);

\* Example to apply the request to every existing process, except the process number 1, with the filter enabled,
	but the override value are not modified in the filter task */
llRetCode	:= F_SetFeedOverride(MODE_NOWAIT, ciProcAll, MI_LastProc, 1 \*iiNoProc*/, liOverride, true \*iOpConsole*/, false \*iOpAdjust*/);
*)

	#IMPORT  "GvU_Variable.gvl"
	#IMPORT  "Gv_Allprocess.gvl"

VAR_INPUT
	iiProc		: int;	(* Process number 1..24 or -1 (ciProcAll) to request to all processes *)
	iiPercent	: int;	(* New override value 10000=100% *)
	iOpConsole	: bool;	(* Console flag, the request is comparable to an operator console, can be rfeused by filter task *)
	iOpAdjust	: bool;	(* Enable modification (Adjust) of override value from PLC request *)
END_VAR

VAR
	llExecStatus	: dword;	(* Function block execution status, not used *)
END_VAR;

gPlcConOvrF[iiProc]	:= iOpConsole;	(* Plc console ambient memory *)
gPlcConAdjF[iiProc]	:= iOpAdjust;	(* Enable modification (Adjust) of override value from PLC request *)
F_SetFeedOverride	:= SetFeedOverride(MODE_NOWAIT, llExecStatus, iiProc, iiPercent);

END_FUNCTION

(* ---- F_SetIncJog.st ---- *)
(*[[
    UserText1= "V15.7",
]]*)
FUNCTION F_SetIncJog : DWORD
(*
F ***************************************************************************************
F * File name    : F_SetIncJog.st                                                       *
F * Description  : Set Incremental Jog request from PLC, works like the system function *
F *                block with two more possibility: the request can be applyed to all   *
F *                processes, have one more flag to decide if the request is comparable *
F *                to an operator request (like a console) and can be refused by the    *
F *                filter task.                                                         *
F ***************************************************************************************
F * Product line : OpenControl                                                          *
F * Enviroment   : PLC Application                                                      *
F * Component    :                                                                      *
F *                                                                                     *
F * ----------------------------------------------------------------------------------- *
F *                                                                                     *
F *   Author        date        comments                                                *
F *                                                                                     *
F *   Scapolan      08-02-2017  Function creation                                       *
F *                                                                                     *
F * ----------------------------------------------------------------------------------- *
F *                                                                                     *
F * Input        :  iiProc              INT                                             *
F *                     Process number 1..24 or -1 (ciProcAll) to request to all        *
F *                     processes.                                                      *
F *                                                                                     *
F *                 iiLastProc          INT                                             *
F *                     Last process number, used only if the request is for all        *
F *                     processes.                                                      *
F *                                                                                     *
F *                 iiNoProc            INT                                             *
F *                     Process number to skip if the request is for all processes,     *
F *                     0 to apply to every processes.                                  *
F *                                                                                     *
F *                 idIncLogValue       LREAL                                           *
F *                     New incremental jog value                                       *
F *                                                                                     *
F *                 iOpConsole          BOOL                                            *
F *                     Console flag, the request is comparable to an operator console, *
F *                     can be rfeused by filter task                                   *
F *                                                                                     *
F * Return       :  DWORD                                                               *
F *                     Set Incremental Jog function block return code                  *
F *                                                                                     *
F * Global used  :  gPlcConIJog         array [0..ciMaxProc] of bool                    *
F *                     Set Incremental Jog request from Plc console ambient memory     *
F *                                                                                     *
F ***************************************************************************************

	Example for program use

\* Set Incremental Jog request from PLC, works like the system function block with two more possibility:
	the request can be applyed to all processes, have one more flag to decide if the request
	is comparable to an operator request (like a console) and can be refused by the filter task. */

llRetCode	:= F_SetIncJog(
	iiProc,			\* IN	INT		Process number 1..24 or -1 (ciProcAll) to request to all processes */
	iiLastProc,		\* IN	INT		Last process number, used only if the request is for all processes */
	iiNoProc,		\* IN	INT		Process number to skip if the request is for all processes, 0 to apply to every processes */
	idIncLogValue,	\* IN	LREAL	New incremental jog value */
	iOpConsole);	\* IN	BOOL	Console flag, the request is comparable to an operator console, can be rfeused by filter task */

\* Example to apply the request only at the selected process with the filter enabled, the 2nd and 3rd input data are not used */
llRetCode	:= F_SetIncJog(SI_PROCSEL, MI_LastProc, 0 \*iiNoProc*/, ldNewIncJog, true \*iOpConsole*/);

\* Example to apply the request to every existing process with the filter enabled */
llRetCode	:= F_SetIncJog(ciProcAll, MI_LastProc, 0 \*iiNoProc*/, ldNewIncJog, true \*iOpConsole*/);

\* Example to apply the request to every existing process, except the process number 1, with the filter enabled */
llRetCode	:= F_SetIncJog(ciProcAll, MI_LastProc, 1 \*iiNoProc*/, ldNewIncJog, true \*iOpConsole*/);
*)

	#IMPORT  "GvU_Variable.gvl"
	#IMPORT  "Gv_Allprocess.gvl"

VAR_INPUT
	iiProc			: int;	(* Process number 1..24 or -1 (ciProcAll) to request to all processes *)
	idIncLogValue	:lreal;	(* New incremental jog value *)
	iOpConsole		: bool;	(* Console flag, the request is comparable to an operator console, can be rfeused by filter task *)
END_VAR

VAR
END_VAR;

gPlcConIJog[iiProc]	:= iOpConsole;	(* Plc console ambient memory *)
F_SetIncJog	:= VAR_Write(iiProc, 0 (*Index*), 0 (*NumChar*), 'JOG', idIncLogValue);

END_FUNCTION

(* ---- F_SetManualOverride.st ---- *)
(*[[
    UserText1= "V15.7",
]]*)
FUNCTION F_SetManualOverride : DWORD
(*
F ***************************************************************************************
F * File name    : F_SetManualOverride.st                                               *
F * Description  : Set Manual override request from PLC, works like the system function *
F *                block with three more possibility: the request can be applyed to all *
F *                processes, one flag permit to decide if the request is comparable    *
F *                to an operator request (like a console) and can be refused by the    *
F *                filter task, another flag enable the modification of the override    *
F *                value in the filter task (for example to align at the predefined     *
F *                steps).                                                              *
F ***************************************************************************************
F * Product line : OpenControl                                                          *
F * Enviroment   : PLC Application                                                      *
F * Component    :                                                                      *
F *                                                                                     *
F * ----------------------------------------------------------------------------------- *
F *                                                                                     *
F *   Author        date        comments                                                *
F *                                                                                     *
F *   Scapolan      08-02-17    Function creation                                       *
F *                                                                                     *
F * ----------------------------------------------------------------------------------- *
F *                                                                                     *
F * Input        :  iiExecMode          INT                                             *
F *                     Command execution modality: MODE_NOWAIT, MODE_WAIT              *
F *                                                                                     *
F *                 iiProc              INT                                             *
F *                     Process number 1..24 or -1 (ciProcAll) to request to all        *
F *                     processes.                                                      *
F *                                                                                     *
F *                 iiLastProc          INT                                             *
F *                     Last process number, used only if the request is for all        *
F *                     processes.                                                      *
F *                                                                                     *
F *                 iiNoProc            INT                                             *
F *                     Process number to skip if the request is for all processes,     *
F *                     0 to apply to every processes.                                  *
F *                                                                                     *
F *                 iiPercent           INT                                             *
F *                     New override value 10000=100%                                   *
F *                                                                                     *
F *                 iiDirection         INT                                             *
F *                     New override direction: 0 POSITIVE_DIR, 1 NEGATIVE_DIR          *
F *                                                                                     *
F *                 iiMode              INT                                             *
F *                     Override mode:                                                  *
F *                         0 MFO_INCREMENTAL increase with positive direction,         *
F *                                           decrease with negative direction.         *
F *                         1 MFO_ABSOLUTE modify override value and direction          *
F *                         2 MFO_DIRECTION modify only direction                       *
F *                         3 MFO_PERCENT modifiy only override percent value           *
F *                                                                                     *
F *                 iOpConsole          BOOL                                            *
F *                     Console flag, the request is comparable to an operator console, *
F *                     can be rfeused by filter task                                   *
F *                                                                                     *
F *                 iOpAdjust           BOOL                                            *
F *                     Enable modification (Adjust) of override value from PLC request *
F *                                                                                     *
F * Return       :  DWORD                                                               *
F *                     SetManualOverride function block return code                    *
F *                                                                                     *
F * Global used  :  gPlcConOvrM          array [0..ciMaxProc] of bool                   *
F *                     Set Manual override request from Plc console ambient memory     *
F *                                                                                     *
F *                 gPlcConAdjM          array [0..ciMaxProc] of BOOL                   *
F *                     Enable the modification of the override value in the filter     *
F *                     task (for example to align at the predefined steps)             *
F *                                                                                     *
F ***************************************************************************************

	Example for program use

\* Set Manual override request from PLC, works like the system function block with two more possibility:
	the request can be applyed to all processes, one flag permit to decide if the request is comparable
	to an operator request (like a console) and can be refused by the filter task, another flag enable the
	modification of the override value in the filter task (for example to align at the predefined steps). */

llRetCode	:= F_SetManualOverride(
	iiExecMode,		\* IN	INT		Command execution modality: MODE_NOWAIT, MODE_WAIT */
	iiProc,			\* IN	INT		Process number 1..24 or -1 (ciProcAll) to request to all processes */
	iiLastProc,		\* IN	INT		Last process number, used only if the request is for all processes */
	iiNoProc,		\* IN	INT		Process number to skip if the request is for all processes, 0 to apply to every processes */
	iiPercent,		\* IN	INT		New override value 10000=100% */
	iiDirection		\* IN	INT		New override direction: 0 POSITIVE_DIR, 1 NEGATIVE_DIR */
	iiMode			\* IN	INT		Override mode:
										0 MFO_INCREMENTAL increase with positive direction, decrease with negative direction.
										1 MFO_ABSOLUTE modify override value and direction
										2 MFO_DIRECTION modify only direction
										3 MFO_PERCENT modifiy only override percent value */
	iOpConsole,		\* IN	BOOL	Console flag, the request is comparable to an operator console, can be rfeused by filter task */
	iOpAdjust);		\* IN	BOOL	Enable modification (Adjust) of override value from this PLC request */

\* Example to apply the request only at the selected process with the filter enabled, the 3rd and 4th input data are not used,
	the override value are not modified in the filter task,
	in this example the function block change only the override value and not the direction */
llRetCode	:= F_SetManualOverride(MODE_NOWAIT, SI_PROCSEL, MI_LastProc, 0 \*iiNoProc*/, liOverride,
	0 \*OverrideDirection not used*/, MFO_PERCENT, true \*iOpConsole*/ false \*iOpAdjust*/);

\* Example to apply the request to every existing process with the filter enabled,
	but the override value are not modified in the filter task,
	in this example the function block change only the override value and not the direction */
llRetCode	:= F_SetManualOverride(MODE_NOWAIT, ciProcAll, MI_LastProc, 0 \*iiNoProc*/, liOverride,
	0 \*OverrideDirection not used*/, MFO_PERCENT, true \*iOpConsole*/ false \*iOpAdjust*/);

\* Example to apply the request to every existing process, except the process number 1, with the filter enabled,
	but the override value are not modified in the filter task,
	in this example the function block change only the override value and not the direction */
llRetCode	:= F_SetManualOverride(MODE_NOWAIT, ciProcAll, MI_LastProc, 1 \*iiNoProc*/, liOverride,
	0 \*OverrideDirection not used*/, MFO_PERCENT, true \*iOpConsole*/ false \*iOpAdjust*/);
*)

	#IMPORT  "GvU_Variable.gvl"
	#IMPORT  "Gv_Allprocess.gvl"

VAR_INPUT
	iiProc		: int;	(* Process number 1..24 or -1 (ciProcAll) to request to all processes *)
	iiPercent	: int;	(* New override value 10000=100% *)
	iiDirection	: int;	(* New override direction: 0 POSITIVE_DIR, 1 NEGATIVE_DIR *)
	iiMode		: int;	(* Override mode:
							0 MFO_INCREMENTAL increase with positive direction, decrease with negative direction.
							1 MFO_ABSOLUTE modify override value and direction
							2 MFO_DIRECTION modify only direction
							3 MFO_PERCENT modifiy only override percent value *)
	iOpConsole	: bool;	(* Console flag, the request is comparable to an operator console, can be rfeused by filter task *)
	iOpAdjust	: bool;	(* Enable modification (Adjust) of override value from PLC request *)
END_VAR

VAR
	llExecStatus	: dword;	(* Function block execution status, not used *)
END_VAR;

gPlcConOvrM[iiProc]	:= iOpConsole;	(* Plc console ambient memory *)
gPlcConAdjM[iiProc]	:= iOpAdjust;	(* Enable modification (Adjust) of override value from PLC request *)
F_SetManualOverride	:= SetManualOverride(MODE_NOWAIT, llExecStatus, iiProc, iiPercent, iiDirection, iiMode);

END_FUNCTION

(* ---- F_SetProcessMode.st ---- *)
(*[[
    UserText1= "V15.7",
]]*)
FUNCTION F_SetProcessMode
(*
F ***************************************************************************************
F * File name    : F_SetProcessMode.st                                                  *
F * Description  : Set Process Mode request from PLC, works like the system function    *
F *                block with two more possibility: the request can be applyed to all   *
F *                processes, have one more flag to decide if the request is comparable *
F *                to an operator request (like a console) and can be refused by the    *
F *                filter task.                                                         *
F ***************************************************************************************
F * Product line : OpenControl                                                          *
F * Enviroment   : PLC Application                                                      *
F * Component    :                                                                      *
F *                                                                                     *
F * ----------------------------------------------------------------------------------- *
F *                                                                                     *
F *   Author        date        comments                                                *
F *                                                                                     *
F *   Scapolan      08-02-17    Function creation                                       *
F *                                                                                     *
F * ----------------------------------------------------------------------------------- *
F *                                                                                     *
F * Input        :  ii_Proc              INT                                            *
F *                     Process number 1..24 	 										*
F *                 iiProcessMode       INT                                             *
F *                     Requested process mode                                          *
F *                                                                                     *
F *                 iOpConsole          BOOL                                            *
F *                     Console flag, the request is comparable to an operator console, *
F *                     can be rfeused by filter task                                   *
F *                                                                                     *
F * Global used  :  gPlcConSPM          array [0..ciMaxProc] of bool                    *
F *                     Set Process Mode request from Plc console ambient memory        *
F *                                                                                     *
F ***************************************************************************************

	Example for program use

\* Set Process Mode request from PLC, works like the system function block with two more possibility:
	the request can be applyed to all processes, have one more flag to decide if the request
	is comparable to an operator request (like a console) and can be refused by the filter task. */

llRetCode	:= F_SetProcessMode(
	iiProc,			\* IN	INT		Process number 1..24 or -1 (ciProcAll) to request to all processes */
	iiProcessMode,	\* IN	INT		Requested process mode */
	iOpConsole);	\* IN	BOOL	Console flag, the request is comparable to an operator console, can be rfeused by filter task */

\* Example to apply the request only at the selected process */
llRetCode	:= F_SetProcessMode(ii_proc, liSelMode, false \*iOpConsole*/);

\* Example to apply the request at all the process selected in the station */
llRetCode	:= F_SetProcessMode(ii_proc, liSelMode, false \*iOpConsole*/);
*)

	#IMPORT  "GvU_Variable.gvl"
	#IMPORT  "Gv_Allprocess.gvl"

VAR_INPUT
	ii_Proc			: int;	(* Process number 1..24 or -1 (ciProcAll) to request to all processes *)
	ii_ProcessMode	: int;	(* Requested process mode *)
	i_OpConsole		: bool;	(* Console flag, the request is comparable to an operator console, can be rfeused by filter task *)
END_VAR

VAR
	ll_ExecStatus	: dword;	(* Function block execution status, not used *)
	ll_RetCode		: dword;
END_VAR;

gPlcConSPM[ii_Proc]	:= i_OpConsole;	(* Plc console ambient memory *)
ll_RetCode	:= SetProcessMode(MODE_NOWAIT, ll_ExecStatus, ii_Proc, ii_ProcessMode);

END_FUNCTION
